Fanuc KAREL source: ko00061.KL

-- PROVISIONAL review KL for V1013-1; original PC SHA256 f9af12b1d715239814a11b61d13055f0ffd50bd272848913dbc95e43ea491b8d
-- Incomplete behavior may be omitted. Consult companion uncertainty JSON. Do not deploy.
PROGRAM KO00061
%NOLOCKGROUP
BEGIN
  -- UNRESOLVED_PC offsets 5-12; opcodes 9D,23
  -- UNRESOLVED_PC offsets 17-69; opcodes 27,27,49,7E,AD,27,49,7E,AD,22,31,7E,4A
  -- UNRESOLVED_PC offsets 74-78; opcodes 7F
END KO00061
